# EPICS substitutions: rogueApp/Db/HEReg.substitutions
file FirFiltering.db
{
        {}
}

file HlsProcessor.db
{
        {}
}

file HlsTrigBuffer.db
{
        {}
}

file HlsDataStream.db
{
        {}
}

file HEBase.template
{
	{}
}
